ABB RobotStudio station: Solution_1_Template.rspag

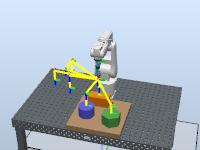
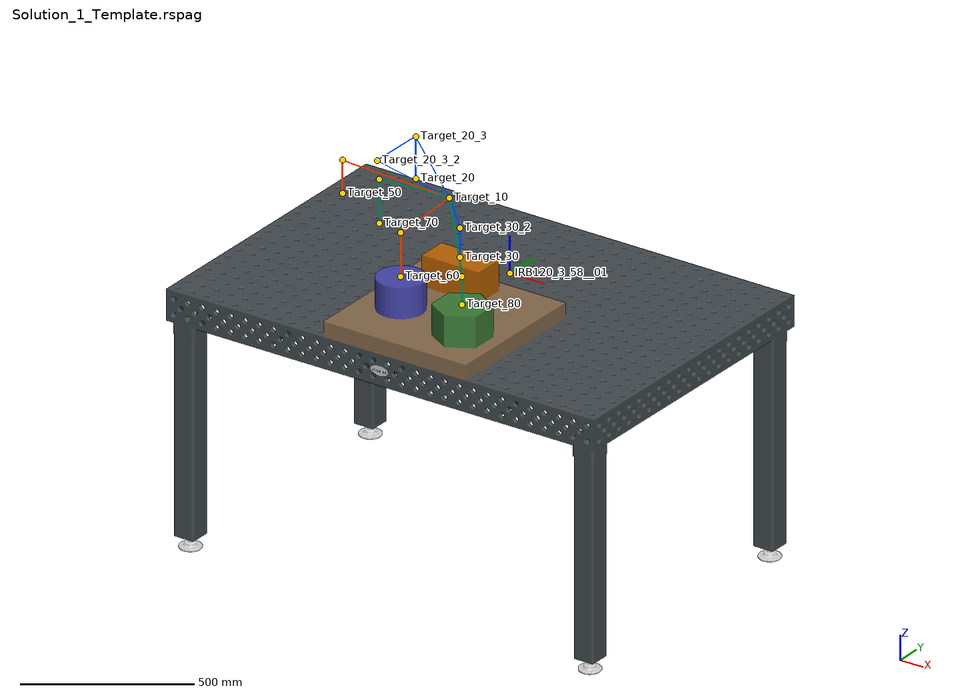
[picture v1: parts stored in the station drawn from their meshes, with robot base, taught points and paths (robot models come from the ABB library and are not in the file)]
--- station ---
Station Solution_1_Tutorial (saved by RobotStudio 21.4.9700.0)
Controller Controller1, task T_ROB1: task frame (RAPID world) sits at (0, 150, 830) mm, rotated rx 0 ry 0 rz -90 deg in the station
Controller Controller1
  mechanical unit ROB_1: IRB120_3_58__01, 6 joints, base frame (0, 0, 0) mm
Layout (positions relative to the parent item):
  - table [part] at (-200, -500, 830) mm, size 500 x 500 x 50 mm
  - object_1 [part] at (-200, -500, 829.92) mm, size 200 x 100 x 150 mm
  - object_2 [part] at (-200, -500, 830.14) mm, size 149.5 x 149.7 x 150 mm
  - object_3 [part] at (-200, -500, 830) mm, size 155.5 x 179.5 x 150 mm
  - siegmund_1500_1000 [part], size 1500 x 1010.3 x 830 mm
  - object_11 [part] at (-200, -500, 830) mm, size 200 x 100 x 150 mm
  - object_22 [part] at (-200, -500, 830) mm, size 149.5 x 149.7 x 150 mm
  - object_33 [part] at (-200, -500, 830) mm, size 155.5 x 179.5 x 150 mm
  - IRB120_3_58__01 [mechanism, from Robots\IRB120_3_58_G_01.rslib] at (0, 150, 830) mm, rotated rx 0 ry 0 rz -90 deg; joint values [0, 0, 0, 0, 1.5708, 0] (rad or m)
  - smc_gripper [mechanism, from 1cv\smc_gripper.rslib] at (0, -152, 1388) mm, rotated rx 180 ry 0 rz 90 deg
  - Attacher_obj_1 [smart component, from Components\Attacher.rslib]
      properties: Parent=smc_gripper; Flange=0; Child=object_1; Mount=false; Offset=[0 0 0]; Orientation=[0 0 0]
  - Detacher_obj_1 [smart component, from Components\Detacher.rslib]
      properties: Child=object_1; KeepPosition=true
  - Attacher_obj_2 [smart component, from Components\Attacher.rslib]
      properties: Parent=smc_gripper; Flange=0; Child=object_2; Mount=false; Offset=[0 0 0]; Orientation=[0 0 0]
  - Detacher_obj_2 [smart component, from Components\Detacher.rslib]
      properties: Child=object_2; KeepPosition=true
  - Positioner_object_3 [smart component, from Components\Positioner.rslib]
      properties: Object=object_3; Position=[-0.7 -0.2 0.83]; Orientation=[0 0 0]; Reference=Global; ReferenceObject=(none)
  - Attacher_obj_3 [smart component, from Components\Attacher.rslib]
      properties: Parent=smc_gripper; Flange=0; Child=object_3; Mount=false; Offset=[0 0 0]; Orientation=[0 0 0]
  - Detacher_obj_3 [smart component, from Components\Detacher.rslib]
      properties: Child=object_3; KeepPosition=true
  - Positioner_object_2 [smart component, from Components\Positioner.rslib]
      properties: Object=object_2; Position=[-0.65 -0.15 0.83]; Orientation=[0 0 0]; Reference=Global; ReferenceObject=(none)
  - Positioner_object_1 [smart component, from Components\Positioner.rslib]
      properties: Object=object_1; Position=[-0.6 -0.15 0.83]; Orientation=[0 0 0]; Reference=Global; ReferenceObject=(none)
Attachment: smc_gripper is attached to IRB120_3_58__01 / Link6
Station signals: DI object_1_positioner, DI object_2_positioner, DI object_3_positioner
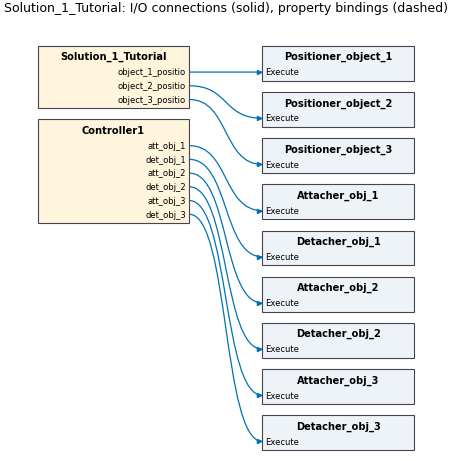
Station logic (signal -> signal, property => property):
  Solution_1_Tutorial.object_1_positioner -> Positioner_object_1.Execute
  Controller1.att_obj_1 -> Attacher_obj_1.Execute
  Controller1.det_obj_1 -> Detacher_obj_1.Execute
  Solution_1_Tutorial.object_2_positioner -> Positioner_object_2.Execute
  Solution_1_Tutorial.object_3_positioner -> Positioner_object_3.Execute
  Controller1.att_obj_2 -> Attacher_obj_2.Execute
  Controller1.det_obj_2 -> Detacher_obj_2.Execute
  Controller1.att_obj_3 -> Attacher_obj_3.Execute
  Controller1.det_obj_3 -> Detacher_obj_3.Execute
Targets, tools, work objects and paths stored in the station and not in the controller backup, written as RAPID:
! task T_ROB1
MODULE Module1
  CONST robtarget Target_40:=[[301.991168121,0.004,360.99899255],[0.000016485,0,-1,0],[-1,-1,-1,0],[9E+09,9E+09,9E+09,9E+09,9E+09,9E+09]];
ENDMODULE


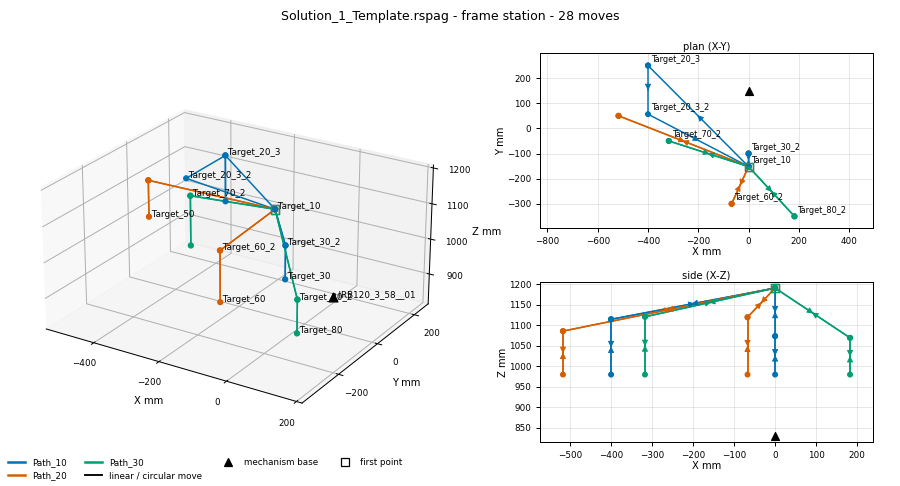
[picture p0: tool path of Solution_1_Template.rspag in frame station, 28 of 28 moves have a stored position in this frame; points joined in program order, loops and branches not executed]
--- Backups/Controller1/RAPID/TASK1/PROGMOD/CalibData.mod ---
MODULE CalibData
    PERS tooldata smc_gripper:=[TRUE,[[0,0.004,197.001],[1,0,0,0]],[1,[0.207,-0.496,71.18],[1,0,0,0],0,0,0]];
ENDMODULE

--- Backups/Controller1/RAPID/TASK1/PROGMOD/Module1.mod ---
MODULE Module1
        CONST robtarget Target_10:=[[301.991141598,0.004,360.999000146],[0.000016466,0,-1,0],[0,0,0,0],[9E+09,9E+09,9E+09,9E+09,9E+09,9E+09]];
    CONST robtarget Target_20_3:=[[-100,-400,284.777898615],[0.000016466,0,-1,0],[-2,-1,-2,0],[9E+09,9E+09,9E+09,9E+09,9E+09,9E+09]];
    CONST robtarget Target_20:=[[-100,-400,150],[0.000016466,0,-1,0],[-2,-1,-2,0],[9E+09,9E+09,9E+09,9E+09,9E+09,9E+09]];
    CONST robtarget Target_30_2:=[[250,0,243.810644535],[0.000016466,0,-1,0],[-1,-1,-1,0],[9E+09,9E+09,9E+09,9E+09,9E+09,9E+09]];
    CONST robtarget Target_30:=[[250,0,150],[0.000016466,0,-1,0],[-1,-1,-1,0],[9E+09,9E+09,9E+09,9E+09,9E+09,9E+09]];
    CONST robtarget Target_50_2:=[[100,-517.298,255.982234266],[0.000016466,0,-1,0],[0,0,0,0],[9E+09,9E+09,9E+09,9E+09,9E+09,9E+09]];
    CONST robtarget Target_50:=[[100,-517.298,150],[0.000016466,0,-1,0],[0,0,0,0],[9E+09,9E+09,9E+09,9E+09,9E+09,9E+09]];
    CONST robtarget Target_60_2:=[[450,-67.298,289.728210899],[0.000016466,0,-1,0],[0,0,0,0],[9E+09,9E+09,9E+09,9E+09,9E+09,9E+09]];
    CONST robtarget Target_60:=[[450,-67.298,150],[0.000016466,0,-1,0],[0,0,0,0],[9E+09,9E+09,9E+09,9E+09,9E+09,9E+09]];
    CONST robtarget Target_70_2:=[[200,-317.298,290.912674672],[0.000016466,0,-1,0],[-1,-1,-1,0],[9E+09,9E+09,9E+09,9E+09,9E+09,9E+09]];
    CONST robtarget Target_70:=[[200,-317.298,150],[0.000016466,0,-1,0],[-1,-1,-1,0],[9E+09,9E+09,9E+09,9E+09,9E+09,9E+09]];
    CONST robtarget Target_80_2:=[[500,182.702,239.605453967],[0.000016466,0,-1,0],[0,0,0,0],[9E+09,9E+09,9E+09,9E+09,9E+09,9E+09]];
    CONST robtarget Target_80:=[[500,182.702,150],[0.000016466,0,-1,0],[0,0,0,0],[9E+09,9E+09,9E+09,9E+09,9E+09,9E+09]];
    CONST robtarget Target_20_3_2:=[[93.581501065,-400,284.777898615],[0.000016466,0,-1,0],[-1,-1,-1,0],[9E+09,9E+09,9E+09,9E+09,9E+09,9E+09]];


    PROC main()
        ! Path 30 -> Pick object 3
        Path_30;
        ! Path 20 -> Pick object 2
        Path_20;
        ! Path 10 -> Pick object 1
        Path_10;
    ENDPROC
    PROC Path_10()
        MoveL Target_10,v200,fine,smc_gripper\WObj:=wobj0;
        MoveL Target_20_3,v200,fine,smc_gripper\WObj:=wobj0;
        MoveL Target_20,v200,fine,smc_gripper\WObj:=wobj0;
        PulseDO att_obj_1;
        WaitTime 1;
        MoveL Target_20_3,v200,fine,smc_gripper\WObj:=wobj0;
        MoveL Target_20_3_2,v200,z100,smc_gripper\WObj:=wobj0;
        MoveL Target_10,v200,fine,smc_gripper\WObj:=wobj0;
        MoveL Target_30_2,v200,fine,smc_gripper\WObj:=wobj0;
        MoveL Target_30,v200,fine,smc_gripper\WObj:=wobj0;
        PulseDO det_obj_1;
        WaitTime 1;
        MoveL Target_30_2,v200,fine,smc_gripper\WObj:=wobj0;
        MoveL Target_10,v200,fine,smc_gripper\WObj:=wobj0;
    ENDPROC
    PROC Path_20()
        MoveL Target_10,v100,fine,smc_gripper\WObj:=wobj0;
        MoveL Target_50_2,v100,fine,smc_gripper\WObj:=wobj0;
        MoveL Target_50,v100,fine,smc_gripper\WObj:=wobj0;
        PulseDO att_obj_2;
        WaitTime 1;
        MoveL Target_50_2,v100,fine,smc_gripper\WObj:=wobj0;
        MoveL Target_10,v100,fine,smc_gripper\WObj:=wobj0;
        MoveL Target_60_2,v100,fine,smc_gripper\WObj:=wobj0;
        MoveL Target_60,v100,fine,smc_gripper\WObj:=wobj0;
        WaitTime 1;
        PulseDO det_obj_2;
        MoveL Target_60_2,v100,fine,smc_gripper\WObj:=wobj0;
        MoveL Target_10,v100,fine,smc_gripper\WObj:=wobj0;
    ENDPROC
    PROC Path_30()
        MoveL Target_10,v150,fine,smc_gripper\WObj:=wobj0;
        MoveL Target_70_2,v150,fine,smc_gripper\WObj:=wobj0;
        MoveL Target_70,v150,fine,smc_gripper\WObj:=wobj0;
        PulseDO att_obj_3;
        WaitTime 1;
        MoveL Target_70_2,v150,fine,smc_gripper\WObj:=wobj0;
        MoveL Target_10,v150,fine,smc_gripper\WObj:=wobj0;
        MoveL Target_80_2,v150,fine,smc_gripper\WObj:=wobj0;
        MoveL Target_80,v150,fine,smc_gripper\WObj:=wobj0;
        PulseDO det_obj_3;
        WaitTime 1;
        MoveL Target_80_2,v150,fine,smc_gripper\WObj:=wobj0;
        MoveL Target_10,v150,fine,smc_gripper\WObj:=wobj0;
    ENDPROC
ENDMODULE

--- Backups/Controller1/SYSPAR/EIO.cfg ---
EIO:CFG_1.0:6:1::
#
EIO_SIGNAL:

      -Name "att_obj_1" -SignalType "DO"

      -Name "det_obj_1" -SignalType "DO"

      -Name "att_obj_2" -SignalType "DO"

      -Name "att_obj_3" -SignalType "DO"

      -Name "det_obj_2" -SignalType "DO"

      -Name "det_obj_3" -SignalType "DO"
